// This function has been automatically generated from the project information.
{attribute 'signature_flag' := '1073741824'}
{attribute 'TcGenerated'}
{attribute 'no-analysis'}
FUNCTION F_GetCompany : WSTRING
VAR_INPUT
	
END_VAR

F_GetCompany := "ekvip automation GmbH";

END_FUNCTION

(* stored: Version 1.1.0.1
   POU F_GetCompany: Id {b319962b-81a0-4689-be82-dd27e14b2082}, SpecialFunc None *)
